SMOVL C01773 BC01773 V=1000.0  +MOVJ EC01773
SMOVL C01774 BC01774 V=1000.0  +MOVJ EC01774
SFTOF3D
'EndPath W4013
'Path W4014
SFTOF3D
SFTON3D P040
MOVJ C01775 BC01775 VJ=100.00  +MOVJ EC01775 VJ=100.00
SMOVL C01776 BC01776 V=800.0  +MOVJ EC01776
SMOVL C01777 BC01777 V=150.0 PL=0  +MOVJ EC01777
ARCON
SMOVL C01778 BC01778 V=10.0  +MOVJ EC01778
ARCOF
SMOVL C01779 BC01779 V=800.0  +MOVJ EC01779
SMOVL C01780 BC01780 V=1000.0  +MOVJ EC01780
SFTOF3D
'EndPath W4014
'
MOVJ C01781 BC01781 VJ=100.00  +MOVJ EC01781 VJ=100.00
MOVJ C01782 BC01782 VJ=100.00  +MOVJ EC01782 VJ=100.00
MOVJ C01783 BC01783 VJ=100.00  +MOVJ EC01783 VJ=100.00
MOVJ C01784 BC01784 VJ=100.00  +MOVJ EC01784 VJ=100.00
MOVJ C01785 BC01785 VJ=100.00  +MOVJ EC01785 VJ=100.00
'Path W3522
SFTOF3D
SFTON3D P045
MOVJ C01786 BC01786 VJ=100.00  +MOVJ EC01786 VJ=100.00
SMOVL C01787 BC01787 V=800.0  +MOVJ EC01787
SMOVL C01788 BC01788 V=150.0 PL=0  +MOVJ EC01788
MACRO1 MJ#(0) ARGF9
ARCON
SMOVL C01789 BC01789 V=11.7  +MOVJ EC01789
ARCOF
SMOVL C01790 BC01790 V=800.0  +MOVJ EC01790
SMOVL C01791 BC01791 V=1000.0  +MOVJ EC01791
SFTOF3D
'EndPath W3522
'Path W3520
SFTOF3D
SFTON3D P044
MOVJ C01792 BC01792 VJ=100.00  +MOVJ EC01792 VJ=100.00
SMOVL C01793 BC01793 V=800.0  +MOVJ EC01793
SMOVL C01794 BC01794 V=166.7 PL=0  +MOVJ EC01794
ARCON
SMOVL C01795 BC01795 V=11.7  +MOVJ EC01795
SMOVL C01796 BC01796 V=11.7  +MOVJ EC01796
SMOVL C01797 BC01797 V=11.7  +MOVJ EC01797
ARCOF
SMOVL C01798 BC01798 V=800.0  +MOVJ EC01798
SMOVL C01799 BC01799 V=1000.0  +MOVJ EC01799
SFTOF3D
'EndPath W3520
'Path W3519
SFTOF3D
SFTON3D P046
MOVJ C01800 BC01800 VJ=100.00  +MOVJ EC01800 VJ=100.00
SMOVL C01801 BC01801 V=800.0  +MOVJ EC01801
SMOVL C01802 BC01802 V=166.7 PL=0  +MOVJ EC01802
ARCON
SMOVL C01803 BC01803 V=12.5  +MOVJ EC01803
SMOVL C01804 BC01804 V=12.5  +MOVJ EC01804
SMOVL C01805 BC01805 V=12.5  +MOVJ EC01805
ARCOF
SMOVL C01806 BC01806 V=800.0  +MOVJ EC01806
SMOVL C01807 BC01807 V=1000.0  +MOVJ EC01807
SFTOF3D
'EndPath W3519
'1
MOVJ C01808 BC01808 VJ=100.00  +MOVJ EC01808 VJ=100.00
MOVJ C01809 BC01809 VJ=100.00  +MOVJ EC01809 VJ=100.00
'Path W3509
SFTOF3D
SFTON3D P048
MOVJ C01810 BC01810 VJ=100.00  +MOVJ EC01810 VJ=100.00
SMOVL C01811 BC01811 V=800.0  +MOVJ EC01811
SMOVL C01812 BC01812 V=150.0 PL=0  +MOVJ EC01812
ARCON
SMOVL C01813 BC01813 V=11.7  +MOVJ EC01813
ARCOF
SMOVL C01814 BC01814 V=800.0  +MOVJ EC01814
SMOVL C01815 BC01815 V=1000.0  +MOVJ EC01815
SFTOF3D
'EndPath W3509
'Path W3510
SFTOF3D
SFTON3D P049
MOVJ C01816 BC01816 VJ=100.00  +MOVJ EC01816 VJ=100.00
SMOVL C01817 BC01817 V=800.0  +MOVJ EC01817
SMOVL C01818 BC01818 V=150.0 PL=0  +MOVJ EC01818
MACRO1 MJ#(0) ARGF6
ARCON
SMOVL C01819 BC01819 V=9.2  +MOVJ EC01819
SMOVL C01820 BC01820 V=9.2  +MOVJ EC01820
SMOVL C01821 BC01821 V=9.2  +MOVJ EC01821
SMOVL C01822 BC01822 V=9.2  +MOVJ EC01822
SMOVL C01823 BC01823 V=9.2  +MOVJ EC01823
ARCOF
MOVJ C01824 BC01824 VJ=30.00  +MOVJ EC01824 VJ=80.00
MOVJ C01825 BC01825 VJ=30.00  +MOVJ EC01825 VJ=30.00
SMOVL C01826 BC01826 V=166.7  +MOVJ EC01826
ARCON
SMOVL C01827 BC01827 V=13.3  +MOVJ EC01827
SMOVL C01828 BC01828 V=13.3  +MOVJ EC01828
SMOVL C01829 BC01829 V=13.3  +MOVJ EC01829
ARCOF
SMOVL C01830 BC01830 V=333.3  +MOVJ EC01830
SMOVL C01831 BC01831 V=666.7  +MOVJ EC01831
SMOVL C01832 BC01832 V=166.7  +MOVJ EC01832
ARCON
SMOVL C01833 BC01833 V=13.3  +MOVJ EC01833
SMOVL C01834 BC01834 V=13.3  +MOVJ EC01834
ARCOF
SMOVL C01835 BC01835 V=166.7  +MOVJ EC01835
ARCON
SMOVL C01836 BC01836 V=11.7  +MOVJ EC01836
ARCOF
SMOVL C01837 BC01837 V=250.0  +MOVJ EC01837
SFTOF3D
'EndPath W3510
MOVJ C01838 BC01838 VJ=100.00  +MOVJ EC01838 VJ=100.00
'2
MOVJ C01839 BC01839 VJ=100.00  +MOVJ EC01839 VJ=100.00
MOVJ C01840 BC01840 VJ=100.00  +MOVJ EC01840 VJ=100.00
MOVJ C01841 BC01841 VJ=100.00  +MOVJ EC01841 VJ=100.00
'Path W3511
SFTOF3D
SFTON3D P043
MOVJ C01842 BC01842 VJ=100.00  +MOVJ EC01842 VJ=100.00
SMOVL C01843 BC01843 V=800.0  +MOVJ EC01843
SMOVL C01844 BC01844 V=166.7 PL=0  +MOVJ EC01844
MACRO1 MJ#(0) ARGF9
ARCON
SMOVL C01845 BC01845 V=11.7  +MOVJ EC01845
ARCOF
SMOVL C01846 BC01846 V=800.0  +MOVJ EC01846
SMOVL C01847 BC01847 V=1000.0  +MOVJ EC01847
SFTOF3D
'EndPath W3511
'Path W3512
SFTOF3D
SFTON3D P042
MOVJ C01848 BC01848 VJ=100.00  +MOVJ EC01848 VJ=100.00
SMOVL C01849 BC01849 V=800.0  +MOVJ EC01849
SMOVL C01850 BC01850 V=150.0 PL=0  +MOVJ EC01850
ARCON
SMOVL C01851 BC01851 V=11.7  +MOVJ EC01851
ARCOF
SMOVL C01852 BC01852 V=800.0  +MOVJ EC01852
SMOVL C01853 BC01853 V=1000.0  +MOVJ EC01853
SFTOF3D
'EndPath W3512
'3
MOVJ C01854 BC01854 VJ=100.00  +MOVJ EC01854 VJ=100.00
MOVJ C01855 BC01855 VJ=100.00  +MOVJ EC01855 VJ=100.00
MOVJ C01856 BC01856 VJ=100.00  +MOVJ EC01856 VJ=100.00
MOVJ C01857 BC01857 VJ=100.00  +MOVJ EC01857 VJ=100.00
'Path W3514
SFTOF3D
SFTON3D P047
MOVJ C01858 BC01858 VJ=100.00  +MOVJ EC01858 VJ=100.00
SMOVL C01859 BC01859 V=800.0  +MOVJ EC01859
SMOVL C01860 BC01860 V=150.0 PL=0  +MOVJ EC01860
ARCON
SMOVL C01861 BC01861 V=11.7  +MOVJ EC01861
ARCOF
SMOVL C01862 BC01862 V=800.0  +MOVJ EC01862
SMOVL C01863 BC01863 V=1000.0  +MOVJ EC01863
SFTOF3D
'EndPath W3514
'Path W3518
SFTOF3D
SFTON3D P047
MOVJ C01864 BC01864 VJ=100.00  +MOVJ EC01864 VJ=100.00
SMOVL C01865 BC01865 V=800.0  +MOVJ EC01865
SMOVL C01866 BC01866 V=150.0 PL=0  +MOVJ EC01866
ARCON
SMOVL C01867 BC01867 V=11.7  +MOVJ EC01867
ARCOF
SMOVL C01868 BC01868 V=800.0  +MOVJ EC01868
SMOVL C01869 BC01869 V=1000.0  +MOVJ EC01869
SFTOF3D
'EndPath W3518
MOVJ C01870 BC01870 VJ=100.00  +MOVJ EC01870 VJ=100.00
MOVJ C01871 BC01871 VJ=100.00  +MOVJ EC01871 VJ=100.00
MOVJ C01872 BC01872 VJ=100.00  +MOVJ EC01872 VJ=100.00
MOVJ C01873 BC01873 VJ=100.00  +MOVJ EC01873 VJ=100.00
'Path W3516
SFTOF3D
SFTON3D P043
MOVJ C01874 BC01874 VJ=50.00  +MOVJ EC01874 VJ=50.00
MOVJ C01875 BC01875 VJ=100.00  +MOVJ EC01875 VJ=100.00
SMOVL C01876 BC01876 V=800.0  +MOVJ EC01876
SMOVL C01877 BC01877 V=150.0 PL=0  +MOVJ EC01877
ARCON
SMOVL C01878 BC01878 V=11.7  +MOVJ EC01878
ARCOF
SMOVL C01879 BC01879 V=800.0  +MOVJ EC01879
SMOVL C01880 BC01880 V=1000.0  +MOVJ EC01880
SFTOF3D
'EndPath W3516
'Path W3515
SFTOF3D
SFTON3D P042
MOVJ C01881 BC01881 VJ=100.00  +MOVJ EC01881 VJ=100.00
SMOVL C01882 BC01882 V=800.0  +MOVJ EC01882
SMOVL C01883 BC01883 V=166.7 PL=0  +MOVJ EC01883
ARCON
SMOVL C01884 BC01884 V=10.8  +MOVJ EC01884
ARCOF
SMOVL C01885 BC01885 V=800.0  +MOVJ EC01885
SMOVL C01886 BC01886 V=1000.0  +MOVJ EC01886
SFTOF3D
'EndPath W3515
MOVJ C01887 BC01887 VJ=100.00  +MOVJ EC01887 VJ=100.00
MOVJ C01888 BC01888 VJ=100.00  +MOVJ EC01888 VJ=100.00
MOVJ C01889 BC01889 VJ=100.00  +MOVJ EC01889 VJ=100.00
MOVJ C01890 BC01890 VJ=100.00  +MOVJ EC01890 VJ=100.00
'Path W3523
SFTOF3D
SFTON3D P046
MOVJ C01891 BC01891 VJ=100.00  +MOVJ EC01891 VJ=100.00
SMOVL C01892 BC01892 V=800.0  +MOVJ EC01892
SMOVL C01893 BC01893 V=166.7 PL=0  +MOVJ EC01893
MACRO1 MJ#(0) ARGF14
ARCON
SMOVL C01894 BC01894 V=10.0  +MOVJ EC01894
ARCOF
SMOVL C01895 BC01895 V=800.0  +MOVJ EC01895
SMOVL C01896 BC01896 V=1000.0  +MOVJ EC01896
SFTOF3D
'EndPath W3523
'Path W4015
SFTOF3D
SFTON3D P044
MOVJ C01897 BC01897 VJ=100.00  +MOVJ EC01897 VJ=100.00
SMOVL C01898 BC01898 V=800.0  +MOVJ EC01898
SMOVL C01899 BC01899 V=150.0 PL=0  +MOVJ EC01899
MACRO1 MJ#(0) ARGF9
ARCON
SMOVL C01900 BC01900 V=10.8  +MOVJ EC01900
ARCOF
SMOVL C01901 BC01901 V=800.0  +MOVJ EC01901
SMOVL C01902 BC01902 V=1000.0  +MOVJ EC01902
SFTOF3D
'EndPath W4015
MOVJ C01903 BC01903 VJ=100.00  +MOVJ EC01903 VJ=100.00
MOVJ C01904 BC01904 VJ=100.00  +MOVJ EC01904 VJ=100.00
MOVJ C01905 BC01905 VJ=100.00  +MOVJ EC01905 VJ=100.00
MOVJ C01906 BC01906 VJ=100.00  +MOVJ EC01906 VJ=100.00
'Path W4016
SFTOF3D
SFTON3D P041
MOVJ C01907 BC01907 VJ=100.00  +MOVJ EC01907 VJ=100.00
SMOVL C01908 BC01908 V=800.0  +MOVJ EC01908
SMOVL C01909 BC01909 V=150.0 PL=0  +MOVJ EC01909
MACRO1 MJ#(0) ARGF14
ARCON
SMOVL C01910 BC01910 V=10.0  +MOVJ EC01910
SMOVL C01911 BC01911 V=10.0  +MOVJ EC01911
SMOVL C01912 BC01912 V=10.0  +MOVJ EC01912
ARCOF
SMOVL C01913 BC01913 V=800.0  +MOVJ EC01913
SMOVL C01914 BC01914 V=1000.0  +MOVJ EC01914
SFTOF3D
'EndPath W4016
'Path W4017
SFTOF3D
SFTON3D P041
MOVJ C01915 BC01915 VJ=100.00  +MOVJ EC01915 VJ=100.00
SMOVL C01916 BC01916 V=800.0  +MOVJ EC01916
SMOVL C01917 BC01917 V=150.0 PL=0  +MOVJ EC01917
COMM SMOVL C01918 BC01918 V=10.0  +MOVJ EC01918
ARCOF
SMOVL C01919 BC01919 V=800.0  +MOVJ EC01919
SMOVL C01920 BC01920 V=1000.0  +MOVJ EC01920
SFTOF3D
'EndPath W4017
MOVJ C01921 BC01921 VJ=100.00  +MOVJ EC01921 VJ=100.00
'Path W4018
SFTOF3D
SFTON3D P041
MOVJ C01922 BC01922 VJ=100.00  +MOVJ EC01922 VJ=100.00
SMOVL C01923 BC01923 V=800.0  +MOVJ EC01923
SMOVL C01924 BC01924 V=150.0 PL=0  +MOVJ EC01924
SMOVL C01925 BC01925 V=10.0  +MOVJ EC01925
ARCOF
SMOVL C01926 BC01926 V=800.0  +MOVJ EC01926
SMOVL C01927 BC01927 V=1000.0  +MOVJ EC01927
SFTOF3D
'EndPath W4018
MOVJ C01928 BC01928 VJ=100.00  +MOVJ EC01928 VJ=100.00
MOVJ C01929 BC01929 VJ=100.00  +MOVJ EC01929 VJ=100.00
MOVJ C01930 BC01930 VJ=100.00  +MOVJ EC01930 VJ=100.00
MOVJ C01931 BC01931 VJ=100.00  +MOVJ EC01931 VJ=100.00
MOVJ C01932 BC01932 VJ=100.00  +MOVJ EC01932 VJ=100.00
END
